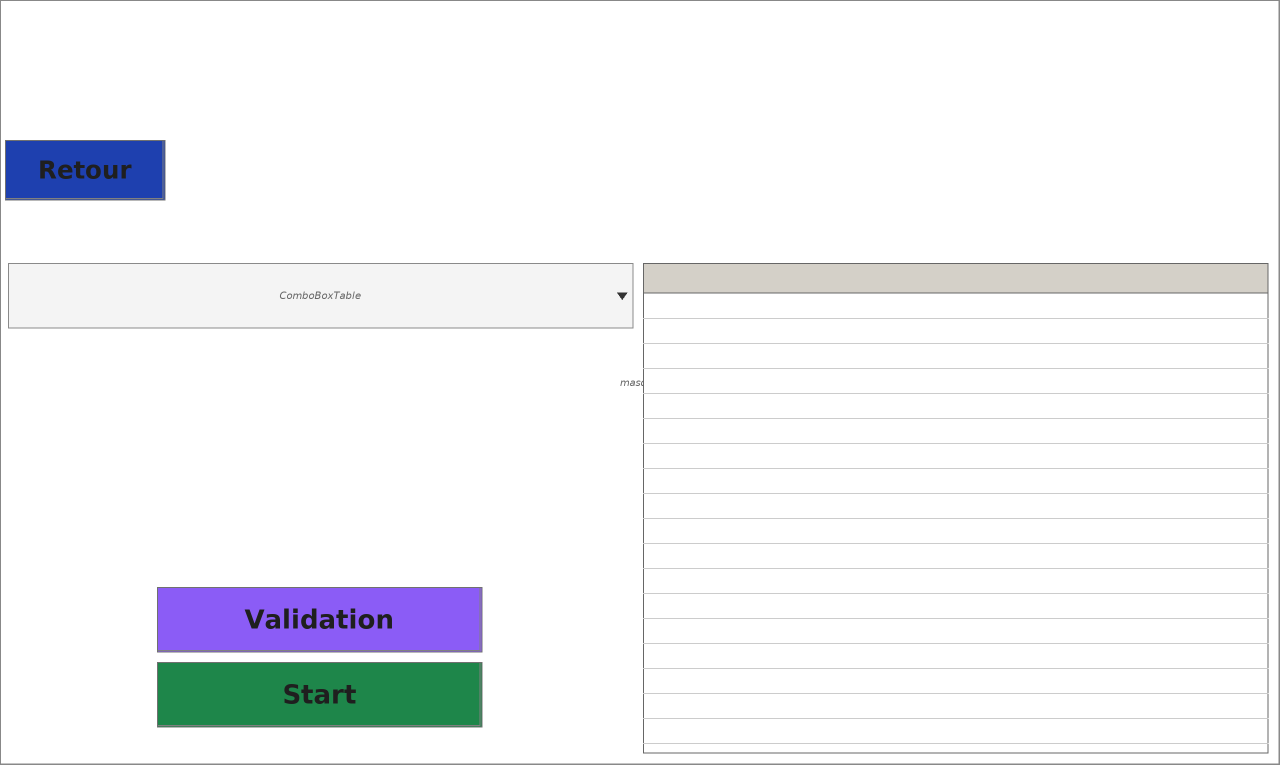
VISUALIZATION Sel_Recettes  // 1280x765
    Frame (0,0 1280x765)
        shows masque()
    ComboBoxTable (8,263 625x65), variable: Numero_Recette_Sel, invisible if: VisuElems.CURRENTLANGUAGE = 'en', data array: Tab_Nom_Recette
        p3854506369: Tab_Nom_Recette[1,INDEX]
        p1892666644: Tab_Nom_Recette[2,INDEX]
    Button (5,140 160x60), "Retour"
        OnMouseDown: change screen: menu
    ComboBoxTable (8,263 625x65), variable: Numero_Recette_Sel, invisible if: VisuElems.CURRENTLANGUAGE = 'fr', data array: Tab_Nom_Recette
        p3854506369: Tab_Nom_Recette[1,INDEX]
        p1892666644: Tab_Nom_Recette[2,INDEX]
    Table (643,263 625x490), invisible if: VisuElems.CURRENTLANGUAGE = 'en', data array: Tab_Nom_Mode
        p3854506369: Tab_Nom_Mode[1,INDEX]
        p1892666644: Tab_Nom_Mode[2,INDEX]
    Rectangle (39,213 562x49), "Veuillez sélectionner une recette", text variable: MES_Debit_Volh_Soufflage
    Rectangle (674,213 562x49), "Détail de la recette sélectionnée", text variable: MES_Debit_Volh_Soufflage
    Table (643,263 625x490), invisible if: VisuElems.CURRENTLANGUAGE = 'fr', data array: Tab_Nom_Mode
        p3854506369: Tab_Nom_Mode[1,INDEX]
        p1892666644: Tab_Nom_Mode[2,INDEX]
    Button (157,587 325x65), "Validation"
        OnMouseDown: toggle Validation_Recette_Auto
    Button (157,662 325x65), "Start", invisible if: GVL_Visu.Visu_Btn_Start
        OnMouseDown: change screen: Recet_EnCours
        OnMouseDown: toggle Start_Recette_Mode_Auto
    RoundedRectangle (118,507 423x65), "Cons. Temp. eau : %.1f °C", text variable: Cons_Temp_EauMitige, invisible if: NOT Option_Regul_Temp_Eau
        OnMouseDown: write the text variable via VisuDialogs.Numpad, min 0, max 50, format %.0f
END_VISUALIZATION

(* stored: Version 1.1.0.1, ProductVersion 3.1.4024.16
   Visu Sel_Recettes: Id {1d41f7cd-5004-49df-8bdf-d3157aebfb8c} *)
